// TIA Portal V20 export
TYPE "typeEm4MonitoringUserDefine"
// stored: Access Published, Namespace Unit1
   STRUCT
      feedingRollJogSpeed { ExternalWritable := 'False'} : LReal;
   END_STRUCT;
END_TYPE
